ABB RAPID module: Module1.mod

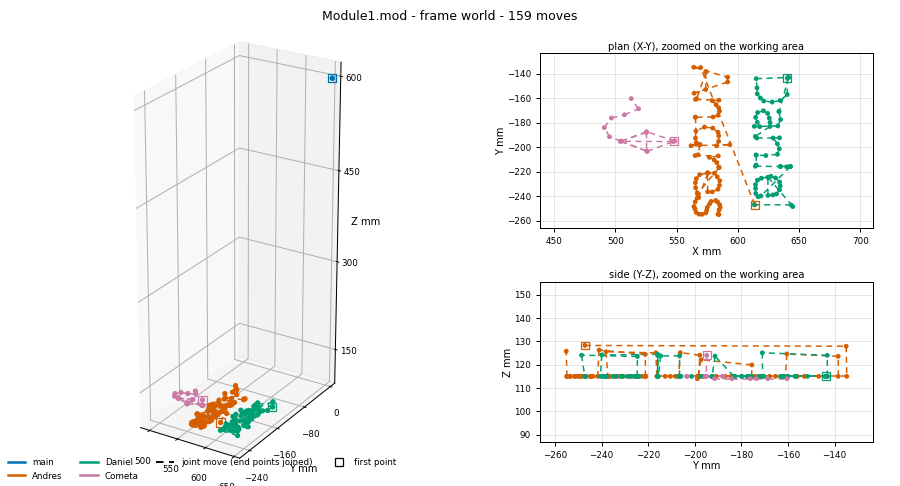
[picture p0: tool path of Module1.mod in frame world, 159 of 159 moves have a stored position in this frame; points joined in program order, loops and branches not executed]
MODULE Module1
    CONST robtarget Target_20:=[[-11.772,36.3,-1],[1,0,0,0],[-1,0,1,0],[9E+09,9E+09,9E+09,9E+09,9E+09,9E+09]];
    CONST robtarget Target_310:=[[-20.078,89.945,-1],[1,0,0,0],[0,0,0,0],[9E+09,9E+09,9E+09,9E+09,9E+09,9E+09]];
    CONST robtarget Target_320:=[[-18.564,93.957,-1],[1,0,0,0],[0,0,0,0],[9E+09,9E+09,9E+09,9E+09,9E+09,9E+09]];
    CONST robtarget Target_330:=[[-20.074,98.498,-1],[1,0,0,0],[0,0,0,0],[9E+09,9E+09,9E+09,9E+09,9E+09,9E+09]];
    CONST robtarget Target_340:=[[-29.523,99.456,-1],[1,0,0,0],[0,0,0,0],[9E+09,9E+09,9E+09,9E+09,9E+09,9E+09]];
    CONST robtarget Target_350:=[[-37.595,99.051,-1],[1,0,0,0],[0,0,0,0],[9E+09,9E+09,9E+09,9E+09,9E+09,9E+09]];
    CONST robtarget Target_360:=[[-37.37,99.043,-9.809],[1,0,0,0],[0,0,0,0],[9E+09,9E+09,9E+09,9E+09,9E+09,9E+09]];
    CONST robtarget Target_370:=[[-37.421,107.137,-9.783],[1,0,0,0],[0,0,0,0],[9E+09,9E+09,9E+09,9E+09,9E+09,9E+09]];
    CONST robtarget Target_10:=[[-30.629,39.059,-159.364],[1,0,0,0],[0,0,0,0],[9E+09,9E+09,9E+09,9E+09,9E+09,9E+09]];
    CONST robtarget Target_60:=[[-31.121,54.924,-1],[1,0,0,0],[-1,0,1,0],[9E+09,9E+09,9E+09,9E+09,9E+09,9E+09]];
    CONST robtarget Target_30:=[[-11.923,49.649,-1],[1,0,0,0],[-1,0,1,0],[9E+09,9E+09,9E+09,9E+09,9E+09,9E+09]];
    CONST robtarget Target_40:=[[-17.688,54.586,-1],[1,0,0,0],[-1,0,1,0],[9E+09,9E+09,9E+09,9E+09,9E+09,9E+09]];
    CONST robtarget Target_50:=[[-24.231,55.786,-1],[1,0,0,0],[-1,0,1,0],[9E+09,9E+09,9E+09,9E+09,9E+09,9E+09]];
    CONST robtarget Target_70:=[[-33.837,52.501,-1],[1,0,0,0],[-1,0,1,0],[9E+09,9E+09,9E+09,9E+09,9E+09,9E+09]];
    CONST robtarget Target_80:=[[-36.393,49.035,-1],[1,0,0,0],[-1,0,1,0],[9E+09,9E+09,9E+09,9E+09,9E+09,9E+09]];
    CONST robtarget Target_90:=[[-36.591,44.152,-1],[1,0,0,0],[-1,0,1,0],[9E+09,9E+09,9E+09,9E+09,9E+09,9E+09]];
    CONST robtarget Target_100:=[[-37.264,36.66,-1],[1,0,0,0],[0,0,0,0],[9E+09,9E+09,9E+09,9E+09,9E+09,9E+09]];
    CONST robtarget Target_110:=[[-11.094,35.738,-1],[1,0,0,0],[0,0,0,0],[9E+09,9E+09,9E+09,9E+09,9E+09,9E+09]];
    CONST robtarget Target_120:=[[-10.813,35.776,-10.021],[1,0,0,0],[0,0,0,0],[9E+09,9E+09,9E+09,9E+09,9E+09,9E+09]];
    CONST robtarget Target_130:=[[-18.604,63.616,-11.122],[1,0,0,0],[0,0,0,0],[9E+09,9E+09,9E+09,9E+09,9E+09,9E+09]];
    CONST robtarget Target_140:=[[-18.774,63.505,-1],[1,0,0,0],[0,0,0,0],[9E+09,9E+09,9E+09,9E+09,9E+09,9E+09]];
    CONST robtarget Target_150:=[[-17.456,70.117,-1],[1,0,0,0],[0,0,0,0],[9E+09,9E+09,9E+09,9E+09,9E+09,9E+09]];
    CONST robtarget Target_160:=[[-19.702,75.325,-1],[1,0,0,0],[0,0,0,0],[9E+09,9E+09,9E+09,9E+09,9E+09,9E+09]];
    CONST robtarget Target_170:=[[-38.911,75.613,-1],[1,0,0,0],[0,0,0,0],[9E+09,9E+09,9E+09,9E+09,9E+09,9E+09]];
    CONST robtarget Target_180:=[[-34.533,75.876,-1],[1,0,0,0],[0,0,0,0],[9E+09,9E+09,9E+09,9E+09,9E+09,9E+09]];
    CONST robtarget Target_190:=[[-36.448,72.308,-1],[1,0,0,0],[0,0,0,0],[9E+09,9E+09,9E+09,9E+09,9E+09,9E+09]];
    CONST robtarget Target_200:=[[-37.782,68.254,-1],[1,0,0,0],[0,0,0,0],[9E+09,9E+09,9E+09,9E+09,9E+09,9E+09]];
    CONST robtarget Target_210:=[[-36.168,64.32,-1],[1,0,0,0],[0,0,0,0],[9E+09,9E+09,9E+09,9E+09,9E+09,9E+09]];
    CONST robtarget Target_220:=[[-31.466,62.883,-1],[1,0,0,0],[0,0,0,0],[9E+09,9E+09,9E+09,9E+09,9E+09,9E+09]];
    CONST robtarget Target_230:=[[-27.942,65.058,-1],[1,0,0,0],[0,0,0,0],[9E+09,9E+09,9E+09,9E+09,9E+09,9E+09]];
    CONST robtarget Target_240:=[[-26.625,68.931,-1],[1,0,0,0],[0,0,0,0],[9E+09,9E+09,9E+09,9E+09,9E+09,9E+09]];
    CONST robtarget Target_250:=[[-26.008,72.574,-1],[1,0,0,0],[0,0,0,0],[9E+09,9E+09,9E+09,9E+09,9E+09,9E+09]];
    CONST robtarget Target_260:=[[-26.244,75.773,-1],[1,0,0,0],[0,0,0,0],[9E+09,9E+09,9E+09,9E+09,9E+09,9E+09]];
    CONST robtarget Target_270:=[[-38.105,83.829,-9.688],[1,0,0,0],[0,0,0,0],[9E+09,9E+09,9E+09,9E+09,9E+09,9E+09]];
    CONST robtarget Target_280:=[[-36.919,85.126,-1],[1,0,0,0],[0,0,0,0],[9E+09,9E+09,9E+09,9E+09,9E+09,9E+09]];
    CONST robtarget Target_290:=[[-18.335,84.993,-1],[1,0,0,0],[0,0,0,0],[9E+09,9E+09,9E+09,9E+09,9E+09,9E+09]];
    CONST robtarget Target_300:=[[-23.583,85.173,-1],[1,0,0,0],[0,0,0,0],[9E+09,9E+09,9E+09,9E+09,9E+09,9E+09]];
    CONST robtarget Target_650:=[[-38.756,139.677,-14.253],[1,0,0,0],[0,0,0,0],[9E+09,9E+09,9E+09,9E+09,9E+09,9E+09]];
    CONST robtarget Target_670:=[[-88.146,27.182,-1],[1,0,0,0],[-1,0,1,0],[9E+09,9E+09,9E+09,9E+09,9E+09,9E+09]];
    CONST robtarget Target_680:=[[-60.482,35.439,-1],[1,0,0,0],[-1,0,1,0],[9E+09,9E+09,9E+09,9E+09,9E+09,9E+09]];
    CONST robtarget Target_690:=[[-60.534,39.292,-1],[1,0,0,0],[-1,0,1,0],[9E+09,9E+09,9E+09,9E+09,9E+09,9E+09]];
    CONST robtarget Target_700:=[[-87.934,48.377,-1],[1,0,0,0],[-1,0,1,0],[9E+09,9E+09,9E+09,9E+09,9E+09,9E+09]];
    CONST robtarget Target_710:=[[-78.498,45.386,-1],[1,0,0,0],[-1,0,1,0],[9E+09,9E+09,9E+09,9E+09,9E+09,9E+09]];
    CONST robtarget Target_720:=[[-78.272,30.843,-1],[1,0,0,0],[-1,0,1,0],[9E+09,9E+09,9E+09,9E+09,9E+09,9E+09]];
    CONST robtarget Target_730:=[[-78.111,30.859,-9.582],[1,0,0,0],[0,0,0,0],[9E+09,9E+09,9E+09,9E+09,9E+09,9E+09]];
    CONST robtarget Target_740:=[[-85.908,52.886,-10.591],[1,0,0,0],[0,0,0,0],[9E+09,9E+09,9E+09,9E+09,9E+09,9E+09]];
    CONST robtarget Target_750:=[[-86.809,53.428,-1],[1,0,0,0],[0,0,0,0],[9E+09,9E+09,9E+09,9E+09,9E+09,9E+09]];
    CONST robtarget Target_760:=[[-67.706,54.137,-1],[1,0,0,0],[0,0,0,0],[9E+09,9E+09,9E+09,9E+09,9E+09,9E+09]];
    CONST robtarget Target_770:=[[-73.231,54.466,-1],[1,0,0,0],[0,0,0,0],[9E+09,9E+09,9E+09,9E+09,9E+09,9E+09]];
    CONST robtarget Target_660:=[[-82.465,27.436,-13.917],[1,0,0,0],[-1,0,1,0],[9E+09,9E+09,9E+09,9E+09,9E+09,9E+09]];
    CONST robtarget Target_380:=[[-38.152,108.13,-1],[1,0,0,0],[0,0,0,0],[9E+09,9E+09,9E+09,9E+09,9E+09,9E+09]];
    CONST robtarget Target_390:=[[-17.806,108.464,-1],[1,0,0,0],[0,0,0,0],[9E+09,9E+09,9E+09,9E+09,9E+09,9E+09]];
    CONST robtarget Target_400:=[[-17.566,108.348,-9.959],[1,0,0,0],[0,0,0,0],[9E+09,9E+09,9E+09,9E+09,9E+09,9E+09]];
    CONST robtarget Target_410:=[[-9.542,108.455,-9.958],[1,0,0,0],[0,0,0,0],[9E+09,9E+09,9E+09,9E+09,9E+09,9E+09]];
    CONST robtarget Target_420:=[[-12.589,108.684,-1],[1,0,0,0],[0,0,0,0],[9E+09,9E+09,9E+09,9E+09,9E+09,9E+09]];
    CONST robtarget Target_430:=[[-9.913,108.523,-1],[1,0,0,0],[0,0,0,0],[9E+09,9E+09,9E+09,9E+09,9E+09,9E+09]];
    CONST robtarget Target_440:=[[-9.515,108.489,-10.438],[1,0,0,0],[0,0,0,0],[9E+09,9E+09,9E+09,9E+09,9E+09,9E+09]];
    CONST robtarget Target_450:=[[-33.66,132.455,-10.194],[1,0,0,0],[0,0,0,0],[9E+09,9E+09,9E+09,9E+09,9E+09,9E+09]];
    CONST robtarget Target_460:=[[-36.019,132.999,-1],[1,0,0,0],[0,0,0,0],[9E+09,9E+09,9E+09,9E+09,9E+09,9E+09]];
    CONST robtarget Target_470:=[[-37.894,130.384,-1],[1,0,0,0],[0,0,0,0],[9E+09,9E+09,9E+09,9E+09,9E+09,9E+09]];
    CONST robtarget Target_480:=[[-38.01,126.323,-1],[1,0,0,0],[0,0,0,0],[9E+09,9E+09,9E+09,9E+09,9E+09,9E+09]];
    CONST robtarget Target_490:=[[-38.113,123.202,-1],[1,0,0,0],[0,0,0,0],[9E+09,9E+09,9E+09,9E+09,9E+09,9E+09]];
    CONST robtarget Target_500:=[[-36.485,119.576,-1],[1,0,0,0],[0,0,0,0],[9E+09,9E+09,9E+09,9E+09,9E+09,9E+09]];
    CONST robtarget Target_510:=[[-33.239,117.955,-1],[1,0,0,0],[0,0,0,0],[9E+09,9E+09,9E+09,9E+09,9E+09,9E+09]];
    CONST robtarget Target_520:=[[-25.533,116.425,-1],[1,0,0,0],[0,0,0,0],[9E+09,9E+09,9E+09,9E+09,9E+09,9E+09]];
    CONST robtarget Target_530:=[[-21.706,117.717,-1],[1,0,0,0],[0,0,0,0],[9E+09,9E+09,9E+09,9E+09,9E+09,9E+09]];
    CONST robtarget Target_540:=[[-18.378,121.103,-1],[1,0,0,0],[0,0,0,0],[9E+09,9E+09,9E+09,9E+09,9E+09,9E+09]];
    CONST robtarget Target_550:=[[-17.916,124.304,-1],[1,0,0,0],[0,0,0,0],[9E+09,9E+09,9E+09,9E+09,9E+09,9E+09]];
    CONST robtarget Target_560:=[[-18.427,127.535,-1],[1,0,0,0],[0,0,0,0],[9E+09,9E+09,9E+09,9E+09,9E+09,9E+09]];
    CONST robtarget Target_570:=[[-20.971,130.791,-1],[1,0,0,0],[0,0,0,0],[9E+09,9E+09,9E+09,9E+09,9E+09,9E+09]];
    CONST robtarget Target_580:=[[-23.95,131.634,-1],[1,0,0,0],[0,0,0,0],[9E+09,9E+09,9E+09,9E+09,9E+09,9E+09]];
    CONST robtarget Target_590:=[[-27.975,132.017,-1],[1,0,0,0],[0,0,0,0],[9E+09,9E+09,9E+09,9E+09,9E+09,9E+09]];
    CONST robtarget Target_600:=[[-27.919,117.225,-1],[1,0,0,0],[0,0,0,0],[9E+09,9E+09,9E+09,9E+09,9E+09,9E+09]];
    CONST robtarget Target_610:=[[-27.772,117.188,-9.546],[1,0,0,0],[0,0,0,0],[9E+09,9E+09,9E+09,9E+09,9E+09,9E+09]];
    CONST robtarget Target_620:=[[-7.716,141.203,-10.062],[1,0,0,0],[0,0,0,0],[9E+09,9E+09,9E+09,9E+09,9E+09,9E+09]];
    CONST robtarget Target_630:=[[-9.032,139.799,-1],[1,0,0,0],[0,0,0,0],[9E+09,9E+09,9E+09,9E+09,9E+09,9E+09]];
    CONST robtarget Target_640:=[[-39.085,139.565,-1],[1,0,0,0],[0,0,0,0],[9E+09,9E+09,9E+09,9E+09,9E+09,9E+09]];
    CONST robtarget Target_800:=[[-67.237,63.087,-1],[1,0,0,0],[0,0,0,0],[9E+09,9E+09,9E+09,9E+09,9E+09,9E+09]];
    CONST robtarget Target_830:=[[-87.101,67.982,-1],[1,0,0,0],[0,0,0,0],[9E+09,9E+09,9E+09,9E+09,9E+09,9E+09]];
    CONST robtarget Target_840:=[[-86.871,67.885,-5.9],[1,0,0,0],[0,0,0,0],[9E+09,9E+09,9E+09,9E+09,9E+09,9E+09]];
    CONST robtarget Target_850:=[[-86.366,89.656,-8.133],[1,0,0,0],[0,0,0,0],[9E+09,9E+09,9E+09,9E+09,9E+09,9E+09]];
    CONST robtarget Target_880:=[[-69.715,91.331,-1],[1,0,0,0],[0,0,0,0],[9E+09,9E+09,9E+09,9E+09,9E+09,9E+09]];
    CONST robtarget Target_890:=[[-68.067,87.731,-1],[1,0,0,0],[0,0,0,0],[9E+09,9E+09,9E+09,9E+09,9E+09,9E+09]];
    CONST robtarget Target_930:=[[-79.521,76.011,-1],[1,0,0,0],[0,0,0,0],[9E+09,9E+09,9E+09,9E+09,9E+09,9E+09]];
    CONST robtarget Target_940:=[[-86.586,79.267,-1],[1,0,0,0],[0,0,0,0],[9E+09,9E+09,9E+09,9E+09,9E+09,9E+09]];
    CONST robtarget Target_950:=[[-87.006,84.957,-1],[1,0,0,0],[0,0,0,0],[9E+09,9E+09,9E+09,9E+09,9E+09,9E+09]];
    CONST robtarget Target_970:=[[-84.038,90.59,-1],[1,0,0,0],[0,0,0,0],[9E+09,9E+09,9E+09,9E+09,9E+09,9E+09]];
    CONST robtarget Target_1000:=[[-87.269,99.259,-1],[1,0,0,0],[0,0,0,0],[9E+09,9E+09,9E+09,9E+09,9E+09,9E+09]];
    CONST robtarget Target_1010:=[[-68.387,99.637,-1],[1,0,0,0],[0,0,0,0],[9E+09,9E+09,9E+09,9E+09,9E+09,9E+09]];
    CONST robtarget Target_1020:=[[-75.689,100.733,-1],[1,0,0,0],[0,0,0,0],[9E+09,9E+09,9E+09,9E+09,9E+09,9E+09]];
    CONST robtarget Target_1030:=[[-71.78,102.882,-1],[1,0,0,0],[0,0,0,0],[9E+09,9E+09,9E+09,9E+09,9E+09,9E+09]];
    CONST robtarget Target_1130:=[[-77.03,113.381,-1],[1,0,0,0],[0,0,0,0],[9E+09,9E+09,9E+09,9E+09,9E+09,9E+09]];
    CONST robtarget Target_1150:=[[-69.289,116.697,-1],[1,0,0,0],[0,0,0,0],[9E+09,9E+09,9E+09,9E+09,9E+09,9E+09]];
    CONST robtarget Target_1170:=[[-67.522,123.662,-1],[1,0,0,0],[0,0,0,0],[9E+09,9E+09,9E+09,9E+09,9E+09,9E+09]];
    CONST robtarget Target_1210:=[[-77.257,113.562,-1],[1,0,0,0],[0,0,0,0],[9E+09,9E+09,9E+09,9E+09,9E+09,9E+09]];
    CONST robtarget Target_1220:=[[-76.871,113.632,-10.411],[1,0,0,0],[0,0,0,0],[9E+09,9E+09,9E+09,9E+09,9E+09,9E+09]];
    CONST robtarget Target_1230:=[[-84.444,133.419,-12.307],[1,0,0,0],[0,0,0,0],[9E+09,9E+09,9E+09,9E+09,9E+09,9E+09]];
    CONST robtarget Target_1240:=[[-85.735,134.036,-1],[1,0,0,0],[0,0,0,0],[9E+09,9E+09,9E+09,9E+09,9E+09,9E+09]];
    CONST robtarget Target_1250:=[[-87.36,137.031,-1],[1,0,0,0],[0,0,0,0],[9E+09,9E+09,9E+09,9E+09,9E+09,9E+09]];
    CONST robtarget Target_1260:=[[-88.386,140.928,-1],[1,0,0,0],[0,0,0,0],[9E+09,9E+09,9E+09,9E+09,9E+09,9E+09]];
    CONST robtarget Target_1280:=[[-86.528,145.651,-1],[1,0,0,0],[0,0,0,0],[9E+09,9E+09,9E+09,9E+09,9E+09,9E+09]];
    CONST robtarget Target_1320:=[[-78.01,143.971,-1],[1,0,0,0],[0,0,0,0],[9E+09,9E+09,9E+09,9E+09,9E+09,9E+09]];
    CONST robtarget Target_1330:=[[-77.462,141.638,-1],[1,0,0,0],[0,0,0,0],[9E+09,9E+09,9E+09,9E+09,9E+09,9E+09]];
    CONST robtarget Target_1340:=[[-75.642,138.894,-1],[1,0,0,0],[0,0,0,0],[9E+09,9E+09,9E+09,9E+09,9E+09,9E+09]];
    CONST robtarget Target_1350:=[[-74.385,136.806,-1],[1,0,0,0],[0,0,0,0],[9E+09,9E+09,9E+09,9E+09,9E+09,9E+09]];
    CONST robtarget Target_1390:=[[-66.977,141.672,-1],[1,0,0,0],[0,0,0,0],[9E+09,9E+09,9E+09,9E+09,9E+09,9E+09]];
    CONST robtarget Target_1400:=[[-67.968,143.816,-1],[1,0,0,0],[0,0,0,0],[9E+09,9E+09,9E+09,9E+09,9E+09,9E+09]];
    CONST robtarget Target_1410:=[[-68.751,147.267,-1],[1,0,0,0],[0,0,0,0],[9E+09,9E+09,9E+09,9E+09,9E+09,9E+09]];
    CONST robtarget Target_1310:=[[-78.714,146.13,-1],[1,0,0,0],[0,0,0,0],[9E+09,9E+09,9E+09,9E+09,9E+09,9E+09]];
    CONST robtarget Target_810:=[[-68.472,66.464,-1],[1,0,0,0],[0,0,0,0],[9E+09,9E+09,9E+09,9E+09,9E+09,9E+09]];
    CONST robtarget Target_1060:=[[-67.657,109.126,-11.089],[1,0,0,0],[0,0,0,0],[9E+09,9E+09,9E+09,9E+09,9E+09,9E+09]];
    CONST robtarget Target_1070:=[[-85.454,130.449,-11.55],[1,0,0,0],[0,0,0,0],[9E+09,9E+09,9E+09,9E+09,9E+09,9E+09]];
    CONST robtarget Target_1190:=[[-73.406,128.984,-1],[1,0,0,0],[0,0,0,0],[9E+09,9E+09,9E+09,9E+09,9E+09,9E+09]];
    CONST robtarget Target_900:=[[-67.972,83.223,-1],[1,0,0,0],[0,0,0,0],[9E+09,9E+09,9E+09,9E+09,9E+09,9E+09]];
    CONST robtarget Target_1420:=[[-68.022,147.553,-11.818],[1,0,0,0],[0,0,0,0],[9E+09,9E+09,9E+09,9E+09,9E+09,9E+09]];
    CONST robtarget Target_1040:=[[-69.558,105.078,-1],[1,0,0,0],[0,0,0,0],[9E+09,9E+09,9E+09,9E+09,9E+09,9E+09]];
    CONST robtarget Target_1270:=[[-87.543,142.809,-1],[1,0,0,0],[0,0,0,0],[9E+09,9E+09,9E+09,9E+09,9E+09,9E+09]];
    CONST robtarget Target_1160:=[[-67.214,119.914,-1],[1,0,0,0],[0,0,0,0],[9E+09,9E+09,9E+09,9E+09,9E+09,9E+09]];
    CONST robtarget Target_1100:=[[-87.158,121.423,-1],[1,0,0,0],[0,0,0,0],[9E+09,9E+09,9E+09,9E+09,9E+09,9E+09]];
    CONST robtarget Target_1360:=[[-70.7,136.052,-1],[1,0,0,0],[0,0,0,0],[9E+09,9E+09,9E+09,9E+09,9E+09,9E+09]];
    CONST robtarget Target_780:=[[-70.054,57.786,-1],[1,0,0,0],[0,0,0,0],[9E+09,9E+09,9E+09,9E+09,9E+09,9E+09]];
    CONST robtarget Target_1080:=[[-85.654,129.675,-1],[1,0,0,0],[0,0,0,0],[9E+09,9E+09,9E+09,9E+09,9E+09,9E+09]];
    CONST robtarget Target_1380:=[[-67.362,139.563,-1],[1,0,0,0],[0,0,0,0],[9E+09,9E+09,9E+09,9E+09,9E+09,9E+09]];
    CONST robtarget Target_820:=[[-72.545,67.817,-1],[1,0,0,0],[0,0,0,0],[9E+09,9E+09,9E+09,9E+09,9E+09,9E+09]];
    CONST robtarget Target_1180:=[[-68.694,126.83,-1],[1,0,0,0],[0,0,0,0],[9E+09,9E+09,9E+09,9E+09,9E+09,9E+09]];
    CONST robtarget Target_1300:=[[-81.685,147.24,-1],[1,0,0,0],[0,0,0,0],[9E+09,9E+09,9E+09,9E+09,9E+09,9E+09]];
    CONST robtarget Target_1140:=[[-71.582,113.745,-1],[1,0,0,0],[0,0,0,0],[9E+09,9E+09,9E+09,9E+09,9E+09,9E+09]];
    CONST robtarget Target_790:=[[-67.904,60.341,-1],[1,0,0,0],[0,0,0,0],[9E+09,9E+09,9E+09,9E+09,9E+09,9E+09]];
    CONST robtarget Target_960:=[[-86.336,88.634,-1],[1,0,0,0],[0,0,0,0],[9E+09,9E+09,9E+09,9E+09,9E+09,9E+09]];
    CONST robtarget Target_1370:=[[-69.086,137.17,-1],[1,0,0,0],[0,0,0,0],[9E+09,9E+09,9E+09,9E+09,9E+09,9E+09]];
    CONST robtarget Target_910:=[[-68.5,80.325,-1],[1,0,0,0],[0,0,0,0],[9E+09,9E+09,9E+09,9E+09,9E+09,9E+09]];
    CONST robtarget Target_1090:=[[-86.972,125.512,-1],[1,0,0,0],[0,0,0,0],[9E+09,9E+09,9E+09,9E+09,9E+09,9E+09]];
    CONST robtarget Target_980:=[[-83.278,90.207,-10.062],[1,0,0,0],[0,0,0,0],[9E+09,9E+09,9E+09,9E+09,9E+09,9E+09]];
    CONST robtarget Target_1200:=[[-77.105,128.829,-1],[1,0,0,0],[0,0,0,0],[9E+09,9E+09,9E+09,9E+09,9E+09,9E+09]];
    CONST robtarget Target_1290:=[[-84.175,147.185,-1],[1,0,0,0],[0,0,0,0],[9E+09,9E+09,9E+09,9E+09,9E+09,9E+09]];
    CONST robtarget Target_1120:=[[-83.667,114.897,-1],[1,0,0,0],[0,0,0,0],[9E+09,9E+09,9E+09,9E+09,9E+09,9E+09]];
    CONST robtarget Target_920:=[[-72.808,76.898,-1],[1,0,0,0],[0,0,0,0],[9E+09,9E+09,9E+09,9E+09,9E+09,9E+09]];
    CONST robtarget Target_1050:=[[-68.061,108.71,-1],[1,0,0,0],[0,0,0,0],[9E+09,9E+09,9E+09,9E+09,9E+09,9E+09]];
    CONST robtarget Target_990:=[[-84.91,98.611,-11.157],[1,0,0,0],[0,0,0,0],[9E+09,9E+09,9E+09,9E+09,9E+09,9E+09]];
    CONST robtarget Target_870:=[[-58.972,90.447,-1],[1,0,0,0],[0,0,0,0],[9E+09,9E+09,9E+09,9E+09,9E+09,9E+09]];
    CONST robtarget Target_860:=[[-90.626,91.24,0],[1,0,0,0],[0,0,0,0],[9E+09,9E+09,9E+09,9E+09,9E+09,9E+09]];
    CONST robtarget Target_1110:=[[-86.368,118.129,-1],[1,0,0,0],[0,0,0,0],[9E+09,9E+09,9E+09,9E+09,9E+09,9E+09]];
    CONST robtarget Target_1430:=[[-104.273,87.192,-10.025],[1,0,0,0],[0,0,0,0],[9E+09,9E+09,9E+09,9E+09,9E+09,9E+09]];
    CONST robtarget Target_1440:=[[-103.744,87.412,-1],[1,0,0,0],[-1,0,1,0],[9E+09,9E+09,9E+09,9E+09,9E+09,9E+09]];
    CONST robtarget Target_1450:=[[-126.812,79.67,-1],[1,0,0,0],[-1,0,1,0],[9E+09,9E+09,9E+09,9E+09,9E+09,9E+09]];
    CONST robtarget Target_1460:=[[-148.382,87.487,-1],[1,0,0,0],[-1,0,1,0],[9E+09,9E+09,9E+09,9E+09,9E+09,9E+09]];
    CONST robtarget Target_1470:=[[-126.39,95.757,-1],[1,0,0,0],[-1,0,1,0],[9E+09,9E+09,9E+09,9E+09,9E+09,9E+09]];
    CONST robtarget Target_1480:=[[-105.403,87.783,-1],[1,0,0,0],[-1,0,1,0],[9E+09,9E+09,9E+09,9E+09,9E+09,9E+09]];
    CONST robtarget Target_1490:=[[-147.834,87.455,-1],[1,0,0,0],[-1,0,1,0],[9E+09,9E+09,9E+09,9E+09,9E+09,9E+09]];
    CONST robtarget Target_1500:=[[-126.956,80.241,-1],[1,0,0,0],[-1,0,1,0],[9E+09,9E+09,9E+09,9E+09,9E+09,9E+09]];
    CONST robtarget Target_1510:=[[-126.868,95.468,-1],[1,0,0,0],[-1,0,1,0],[9E+09,9E+09,9E+09,9E+09,9E+09,9E+09]];
    CONST robtarget Target_1520:=[[-147.679,87.217,-1],[1,0,0,0],[-1,0,1,0],[9E+09,9E+09,9E+09,9E+09,9E+09,9E+09]];
    CONST robtarget Target_1530:=[[-157.131,83.68,0],[1,0,0,0],[-1,0,1,0],[9E+09,9E+09,9E+09,9E+09,9E+09,9E+09]];
    CONST robtarget Target_1540:=[[-161.355,76.172,0],[1,0,0,0],[-1,0,1,0],[9E+09,9E+09,9E+09,9E+09,9E+09,9E+09]];
    CONST robtarget Target_1550:=[[-155.572,68.389,0],[1,0,0,0],[-1,0,1,0],[9E+09,9E+09,9E+09,9E+09,9E+09,9E+09]];
    CONST robtarget Target_1560:=[[-144.829,65.777,0],[1,0,0,0],[-1,0,1,0],[9E+09,9E+09,9E+09,9E+09,9E+09,9E+09]];
    CONST robtarget Target_1570:=[[-133.354,60.946,0],[1,0,0,0],[0,0,0,0],[9E+09,9E+09,9E+09,9E+09,9E+09,9E+09]];
    CONST robtarget Target_1590:=[[-125.401,95.165,-149.148],[1,0,0,0],[0,0,0,0],[9E+09,9E+09,9E+09,9E+09,9E+09,9E+09]];
    CONST robtarget Target_1580:=[[-139.33,52.599,0],[1,0,0,0],[0,0,0,0],[9E+09,9E+09,9E+09,9E+09,9E+09,9E+09]];
    PERS tooldata Marcador:=[TRUE,[[0,0,180],[1,0,0,0]],[1,[0,0,1],[1,0,0,0],0,0,0]];
    TASK PERS wobjdata Workobject_1:=[FALSE,TRUE,"",[[652.068,-107.373,114],[0,0.999998666,0.001633441,0]],[[0,0,0],[1,0,0,0]]];
    CONST robtarget Home_10:=[[652.073,1.754,599.195],[0.5,0,0.866025404,0],[0,0,0,0],[9E+09,9E+09,9E+09,9E+09,9E+09,9E+09]];
!***********************************************************
    !
    ! Módulo:  Module1
    !
    ! Descripción:
    !   <Introduzca la descripción aquí>
    !
    ! Autor: Juan
    !
    ! Versión: 1.0
    !
    !***********************************************************


    !***********************************************************
    !
    ! Procedimiento Main
    !
    !   Este es el punto de entrada de su programa
    !
    !***********************************************************
    PROC main()
        !Añada aquí su código
        MoveJ Home_10,v500,z100,Marcador\WObj:=wobj0;
        Daniel;
        Andres;
        Cometa;
        MoveJ Home_10,v500,z100,Marcador\WObj:=wobj0;
    ENDPROC
    PROC Andres()
        MoveJ Target_650,v100,z100,Marcador\WObj:=Workobject_1;
        MoveJ Target_660,v100,z100,Marcador\WObj:=Workobject_1;
        MoveJ Target_670,v100,z100,Marcador\WObj:=Workobject_1;
        MoveJ Target_680,v100,z100,Marcador\WObj:=Workobject_1;
        MoveJ Target_690,v100,z100,Marcador\WObj:=Workobject_1;
        MoveJ Target_700,v100,z100,Marcador\WObj:=Workobject_1;
        MoveJ Target_710,v100,z100,Marcador\WObj:=Workobject_1;
        MoveJ Target_720,v100,z100,Marcador\WObj:=Workobject_1;
        MoveJ Target_730,v100,z100,Marcador\WObj:=Workobject_1;
        MoveJ Target_740,v100,z100,Marcador\WObj:=Workobject_1;
        MoveJ Target_750,v100,z100,Marcador\WObj:=Workobject_1;
        MoveJ Target_760,v100,z100,Marcador\WObj:=Workobject_1;
        MoveJ Target_770,v100,z100,Marcador\WObj:=Workobject_1;
        MoveJ Target_780,v100,z100,Marcador\WObj:=Workobject_1;
        MoveJ Target_790,v100,z100,Marcador\WObj:=Workobject_1;
        MoveJ Target_800,v100,z100,Marcador\WObj:=Workobject_1;
        MoveJ Target_810,v100,z100,Marcador\WObj:=Workobject_1;
        MoveJ Target_820,v100,z100,Marcador\WObj:=Workobject_1;
        MoveJ Target_830,v100,z100,Marcador\WObj:=Workobject_1;
        MoveJ Target_840,v100,z100,Marcador\WObj:=Workobject_1;
        MoveJ Target_850,v100,z100,Marcador\WObj:=Workobject_1;
        MoveJ Target_860,v100,z100,Marcador\WObj:=Workobject_1;
        MoveJ Target_870,v100,z100,Marcador\WObj:=Workobject_1;
        MoveJ Target_880,v100,z100,Marcador\WObj:=Workobject_1;
        MoveJ Target_890,v100,z100,Marcador\WObj:=Workobject_1;
        MoveJ Target_900,v100,z100,Marcador\WObj:=Workobject_1;
        MoveJ Target_910,v100,z100,Marcador\WObj:=Workobject_1;
        MoveJ Target_920,v100,z100,Marcador\WObj:=Workobject_1;
        MoveJ Target_930,v100,z100,Marcador\WObj:=Workobject_1;
        MoveJ Target_940,v100,z100,Marcador\WObj:=Workobject_1;
        MoveJ Target_950,v100,z100,Marcador\WObj:=Workobject_1;
        MoveJ Target_960,v100,z100,Marcador\WObj:=Workobject_1;
        MoveJ Target_970,v100,z100,Marcador\WObj:=Workobject_1;
        MoveJ Target_980,v100,z100,Marcador\WObj:=Workobject_1;
        MoveJ Target_990,v100,z100,Marcador\WObj:=Workobject_1;
        MoveJ Target_1000,v100,z100,Marcador\WObj:=Workobject_1;
        MoveJ Target_1010,v100,z100,Marcador\WObj:=Workobject_1;
        MoveJ Target_1020,v100,z100,Marcador\WObj:=Workobject_1;
        MoveJ Target_1030,v100,z100,Marcador\WObj:=Workobject_1;
        MoveJ Target_1040,v100,z100,Marcador\WObj:=Workobject_1;
        MoveJ Target_1050,v100,z100,Marcador\WObj:=Workobject_1;
        MoveJ Target_1060,v100,z100,Marcador\WObj:=Workobject_1;
        MoveJ Target_1070,v100,z100,Marcador\WObj:=Workobject_1;
        MoveJ Target_1080,v100,z100,Marcador\WObj:=Workobject_1;
        MoveJ Target_1090,v100,z100,Marcador\WObj:=Workobject_1;
        MoveJ Target_1100,v100,z100,Marcador\WObj:=Workobject_1;
        MoveJ Target_1110,v100,z100,Marcador\WObj:=Workobject_1;
        MoveJ Target_1120,v100,z100,Marcador\WObj:=Workobject_1;
        MoveJ Target_1130,v100,z100,Marcador\WObj:=Workobject_1;
        MoveJ Target_1140,v100,z100,Marcador\WObj:=Workobject_1;
        MoveJ Target_1150,v100,z100,Marcador\WObj:=Workobject_1;
        MoveJ Target_1160,v100,z100,Marcador\WObj:=Workobject_1;
        MoveJ Target_1170,v100,z100,Marcador\WObj:=Workobject_1;
        MoveJ Target_1180,v100,z100,Marcador\WObj:=Workobject_1;
        MoveJ Target_1190,v100,z100,Marcador\WObj:=Workobject_1;
        MoveJ Target_1200,v100,z100,Marcador\WObj:=Workobject_1;
        MoveJ Target_1210,v100,z100,Marcador\WObj:=Workobject_1;
        MoveJ Target_1220,v100,z100,Marcador\WObj:=Workobject_1;
        MoveJ Target_1230,v100,z100,Marcador\WObj:=Workobject_1;
        MoveJ Target_1240,v100,z100,Marcador\WObj:=Workobject_1;
        MoveJ Target_1250,v100,z100,Marcador\WObj:=Workobject_1;
        MoveJ Target_1260,v100,z100,Marcador\WObj:=Workobject_1;
        MoveJ Target_1270,v100,z100,Marcador\WObj:=Workobject_1;
        MoveJ Target_1280,v100,z100,Marcador\WObj:=Workobject_1;
        MoveJ Target_1290,v100,z100,Marcador\WObj:=Workobject_1;
        MoveJ Target_1300,v100,z100,Marcador\WObj:=Workobject_1;
        MoveJ Target_1310,v100,z100,Marcador\WObj:=Workobject_1;
        MoveJ Target_1320,v100,z100,Marcador\WObj:=Workobject_1;
        MoveJ Target_1330,v100,z100,Marcador\WObj:=Workobject_1;
        MoveJ Target_1340,v100,z100,Marcador\WObj:=Workobject_1;
        MoveJ Target_1350,v100,z100,Marcador\WObj:=Workobject_1;
        MoveJ Target_1360,v100,z100,Marcador\WObj:=Workobject_1;
        MoveJ Target_1370,v100,z100,Marcador\WObj:=Workobject_1;
        MoveJ Target_1380,v100,z100,Marcador\WObj:=Workobject_1;
        MoveJ Target_1390,v100,z100,Marcador\WObj:=Workobject_1;
        MoveJ Target_1400,v100,z100,Marcador\WObj:=Workobject_1;
        MoveJ Target_1410,v100,z100,Marcador\WObj:=Workobject_1;
        MoveJ Target_1420,v100,z100,Marcador\WObj:=Workobject_1;
    ENDPROC
    PROC Daniel()
        MoveJ Target_20,v100,z100,Marcador\WObj:=Workobject_1;
        MoveJ Target_30,v100,z100,Marcador\WObj:=Workobject_1;
        MoveJ Target_40,v100,z100,Marcador\WObj:=Workobject_1;
        MoveJ Target_50,v100,z100,Marcador\WObj:=Workobject_1;
        MoveJ Target_60,v100,z100,Marcador\WObj:=Workobject_1;
        MoveJ Target_70,v100,z100,Marcador\WObj:=Workobject_1;
        MoveJ Target_80,v100,z100,Marcador\WObj:=Workobject_1;
        MoveJ Target_90,v100,z100,Marcador\WObj:=Workobject_1;
        MoveJ Target_100,v100,z100,Marcador\WObj:=Workobject_1;
        MoveJ Target_110,v100,z100,Marcador\WObj:=Workobject_1;
        MoveJ Target_120,v100,z100,Marcador\WObj:=Workobject_1;
        MoveJ Target_130,v100,z100,Marcador\WObj:=Workobject_1;
        MoveJ Target_140,v100,z100,Marcador\WObj:=Workobject_1;
        MoveJ Target_150,v100,z100,Marcador\WObj:=Workobject_1;
        MoveJ Target_160,v100,z100,Marcador\WObj:=Workobject_1;
        MoveJ Target_170,v100,z100,Marcador\WObj:=Workobject_1;
        MoveJ Target_180,v100,z100,Marcador\WObj:=Workobject_1;
        MoveJ Target_190,v100,z100,Marcador\WObj:=Workobject_1;
        MoveJ Target_200,v100,z100,Marcador\WObj:=Workobject_1;
        MoveJ Target_210,v100,z100,Marcador\WObj:=Workobject_1;
        MoveJ Target_220,v100,z100,Marcador\WObj:=Workobject_1;
        MoveJ Target_230,v100,z100,Marcador\WObj:=Workobject_1;
        MoveJ Target_240,v100,z100,Marcador\WObj:=Workobject_1;
        MoveJ Target_250,v100,z100,Marcador\WObj:=Workobject_1;
        MoveJ Target_260,v100,z100,Marcador\WObj:=Workobject_1;
        MoveJ Target_270,v100,z100,Marcador\WObj:=Workobject_1;
        MoveJ Target_280,v100,z100,Marcador\WObj:=Workobject_1;
        MoveJ Target_290,v100,z100,Marcador\WObj:=Workobject_1;
        MoveJ Target_300,v100,z100,Marcador\WObj:=Workobject_1;
        MoveJ Target_310,v100,z100,Marcador\WObj:=Workobject_1;
        MoveJ Target_320,v100,z100,Marcador\WObj:=Workobject_1;
        MoveJ Target_330,v100,z100,Marcador\WObj:=Workobject_1;
        MoveJ Target_340,v100,z100,Marcador\WObj:=Workobject_1;
        MoveJ Target_350,v100,z100,Marcador\WObj:=Workobject_1;
        MoveJ Target_360,v100,z100,Marcador\WObj:=Workobject_1;
        MoveJ Target_370,v100,z100,Marcador\WObj:=Workobject_1;
        MoveJ Target_380,v100,z100,Marcador\WObj:=Workobject_1;
        MoveJ Target_390,v100,z100,Marcador\WObj:=Workobject_1;
        MoveJ Target_400,v100,z100,Marcador\WObj:=Workobject_1;
        MoveJ Target_410,v100,z100,Marcador\WObj:=Workobject_1;
        MoveJ Target_420,v100,z100,Marcador\WObj:=Workobject_1;
        MoveJ Target_430,v100,z100,Marcador\WObj:=Workobject_1;
        MoveJ Target_440,v100,z100,Marcador\WObj:=Workobject_1;
        MoveJ Target_450,v100,z100,Marcador\WObj:=Workobject_1;
        MoveJ Target_460,v100,z100,Marcador\WObj:=Workobject_1;
        MoveJ Target_470,v100,z100,Marcador\WObj:=Workobject_1;
        MoveJ Target_480,v100,z100,Marcador\WObj:=Workobject_1;
        MoveJ Target_490,v100,z100,Marcador\WObj:=Workobject_1;
        MoveJ Target_500,v100,z100,Marcador\WObj:=Workobject_1;
        MoveJ Target_510,v100,z100,Marcador\WObj:=Workobject_1;
        MoveJ Target_520,v100,z100,Marcador\WObj:=Workobject_1;
        MoveJ Target_530,v100,z100,Marcador\WObj:=Workobject_1;
        MoveJ Target_540,v100,z100,Marcador\WObj:=Workobject_1;
        MoveJ Target_550,v100,z100,Marcador\WObj:=Workobject_1;
        MoveJ Target_560,v100,z100,Marcador\WObj:=Workobject_1;
        MoveJ Target_570,v100,z100,Marcador\WObj:=Workobject_1;
        MoveJ Target_580,v100,z100,Marcador\WObj:=Workobject_1;
        MoveJ Target_590,v100,z100,Marcador\WObj:=Workobject_1;
        MoveJ Target_600,v100,z100,Marcador\WObj:=Workobject_1;
        MoveJ Target_610,v100,z100,Marcador\WObj:=Workobject_1;
        MoveJ Target_620,v100,z100,Marcador\WObj:=Workobject_1;
        MoveJ Target_630,v100,z100,Marcador\WObj:=Workobject_1;
        MoveJ Target_640,v100,z100,Marcador\WObj:=Workobject_1;
    ENDPROC
    PROC Cometa()
        MoveJ Target_1430,v100,z100,Marcador\WObj:=Workobject_1;
        MoveJ Target_1440,v100,z100,Marcador\WObj:=Workobject_1;
        MoveJ Target_1450,v100,z100,Marcador\WObj:=Workobject_1;
        MoveJ Target_1460,v100,z100,Marcador\WObj:=Workobject_1;
        MoveJ Target_1470,v100,z100,Marcador\WObj:=Workobject_1;
        MoveJ Target_1480,v100,z100,Marcador\WObj:=Workobject_1;
        MoveJ Target_1490,v100,z100,Marcador\WObj:=Workobject_1;
        MoveJ Target_1500,v100,z100,Marcador\WObj:=Workobject_1;
        MoveJ Target_1510,v100,z100,Marcador\WObj:=Workobject_1;
        MoveJ Target_1520,v100,z100,Marcador\WObj:=Workobject_1;
        MoveJ Target_1530,v100,z100,Marcador\WObj:=Workobject_1;
        MoveJ Target_1540,v100,z100,Marcador\WObj:=Workobject_1;
        MoveJ Target_1550,v100,z100,Marcador\WObj:=Workobject_1;
        MoveJ Target_1560,v100,z100,Marcador\WObj:=Workobject_1;
        MoveJ Target_1570,v100,z100,Marcador\WObj:=Workobject_1;
        MoveJ Target_1580,v100,z100,Marcador\WObj:=Workobject_1;
    ENDPROC
ENDMODULE
